// TIA Portal V20 export
DATA_BLOCK "Max_Min_Temp_DB"   // DB58
// stored: InstanceOfName Max_Min_Temp, InstanceOfType FB
"Max_Min_Temp"
   // VAR_INPUT
   //    TempCur : Real;
   // END_VAR
   // VAR_OUTPUT
   //    MaxTemp : Real;
   //    MinTemp : Real;
   // END_VAR
BEGIN
END_DATA_BLOCK
